// TwinCAT 3 PLC project PLC_2
// ProgramVersion: 3.1.4020.2
// libraries:
//   Tc2_Standard, * (Beckhoff Automation GmbH)
//   Tc2_System, * (Beckhoff Automation GmbH)
//   Tc3_Module, * (Beckhoff Automation GmbH)
// project tree:
//   DUTs/ PALLET.TcDUT
//   / GlobalTextList.TcGTLO, PlcTask.TcTTO, Visualization Manager.TcVMO (not stored)
//   POUs/ MAIN.TcPOU
//   VISUs/ Visualization.TcVIS
// real-time tasks:
//   TASK PlcTask: cycle T#10ms, priority 20, ADS port 350

CONFIGURATION PLC_2
    RESOURCE PLC ON TwinCAT3
        TASK PlcTask(INTERVAL := T#10ms, PRIORITY := 20);
        PROGRAM MAIN WITH PlcTask : MAIN;
    END_RESOURCE
END_CONFIGURATION

// ---- DUTs/PALLET.TcDUT
TYPE PALLET :
STRUCT
	EX : BOOL:=FALSE;
	WS2 : BOOL:=FALSE;
	WS3 : BOOL:=FALSE;
	POSITION : INT:=-1;
	NEXT_PALLET : INT:=0;
	PREVIOUS_PALLET : INT:=0;
	NUMBER : INT;
END_STRUCT
END_TYPE

// ---- POUs/MAIN.TcPOU
PROGRAM MAIN
VAR

PALLETS : ARRAY [1..50] OF PALLET;					// array that will contain the pallet's information. The number of pallets is limitted by 50 but the code work for as many pallets as we want.
INDEX_PALLET : ARRAY [1..50] OF INT := [50(50)];	// array that will contain the index of each pallet in the PALLETS array
NUMBER_PALLETS : ARRAY [1..9] OF INT;				// number of pallets in every possible position of the system

// Inputs
START : BOOL;
P1 : BOOL;
P2 : BOOL;
P3 : BOOL;
L1 : BOOL;
L2 : BOOL;
L3 : BOOL;
PALLET_IN : BOOL;

// Outputs
BA1 : BOOL;
BA2 : BOOL;
BA3 : BOOL;
S1 : BOOL:=TRUE;
S2 : BOOL:=TRUE;
S3 : BOOL:=TRUE;


MOTOR : BOOL;			// Motor signal
COUNTER_IN : INT:=0;	// number of pallets that have been introduced to the system
COUNTER_OUT : INT:=0;	// number of pallets that have been processed by all of th workstation

// Auxiliary variables
STATE_OUT : INT:=0;			
f : INT;
PROCESS_COUNTER_OUT : TON;	// timer 5s
COUNTER_WS2 : TON;			// timer 5s
COUNTER_WS3 : TON;			// timer 5s
COUNTER_PICK2 : TON;		// timer 2s for picking up pallets from conveyor to workstation 2 and timer for letting pallet pass through the stopper 2
COUNTER_PICK3 : TON;		// timer 2s. The same as COUNTER_PICK2 but for workstation 3
COUNTER_PICK1 : TON;		// timer 2s. The same as COUNTER_PICK2 but for workstation 1
POSITION2 : BOOL;			// variable that will indicate that a pallet is in front of workstation 2
POSITION3 : BOOL;			// variable that will indicate that a pallet is in front of workstation 3
POSITION1 : BOOL;			// variable that will indicate that a pallet is in front of workstation 1
INDEX : INT;				// index of the last pallet inside the system

END_VAR


// External states 0, 1, 2 and 3
CASE STATE_OUT OF
	0:
	// state that means that the system is not working
	IF START=TRUE THEN
		STATE_OUT:=1;
		MOTOR:= 1;
	END_IF
	1:
	// system is runing. If we insert a pallet, this state is going to insert the pallet in the system
	IF PALLET_IN=TRUE AND NOT L1 THEN
		STATE_OUT:=2;		
		COUNTER_IN:=COUNTER_IN+1;		
		IF (COUNTER_IN-COUNTER_OUT)>1 THEN
			PALLETS[INDEX].NEXT_PALLET := (COUNTER_IN-COUNTER_OUT);
			PALLETS[(COUNTER_IN-COUNTER_OUT)].NEXT_PALLET :=0;
			PALLETS[(COUNTER_IN-COUNTER_OUT)].PREVIOUS_PALLET :=INDEX;			
		END_IF
		L1:=TRUE;
		PALLET_IN:=FALSE;
		PROCESS_COUNTER_OUT(IN:=FALSE, PT :=T#5S);
	END_IF
	IF PALLET_IN AND L1 THEN
		STATE_OUT:=3;
	END_IF
	
	2:
	// when a pallet is inserted, she is inserted in workstation 1 and this workstation start by processing the pallet. This takes 5 seconds
	PROCESS_COUNTER_OUT(IN:=TRUE, PT :=T#5S);
	IF PROCESS_COUNTER_OUT.Q THEN
		STATE_OUT:=3;
		L1:=FALSE;
		INDEX_PALLET[COUNTER_IN]:=COUNTER_IN-COUNTER_OUT;
		NUMBER_PALLETS[1]:=NUMBER_PALLETS[1]+1;
		PALLETS[(COUNTER_IN-COUNTER_OUT)].POSITION :=0;
		PALLETS[(COUNTER_IN-COUNTER_OUT)].EX :=TRUE;
		PALLETS[(COUNTER_IN-COUNTER_OUT)].NUMBER :=COUNTER_IN;
	END_IF
	
	3:
	// in this state, the system will pass through all of the pallets that are in the system. He will see where are they and, depending on the inputs, he will do something to the pallets.
	IF PALLET_IN THEN
		// if PALLETS_IN is pressed, then we have to jump to external state 1 to insert the pallet.
		STATE_OUT:=1;	
	END_IF	
	
	// these nex lines of code exist to find the pallet that is in the front of all of them
	IF PALLETS[1].PREVIOUS_PALLET>0 THEN
		f:=1;
		WHILE PALLETS[f].PREVIOUS_PALLET>0 DO
			f:=PALLETS[f].PREVIOUS_PALLET;
		END_WHILE
	ELSE
		f:=1;
	END_IF	
	
	// WHILE cycle, where the system will pass through all of the pallets in the system
	WHILE f>0 DO
		INDEX:=f;
		// Internal states
		CASE PALLETS[f].POSITION OF
			0:
			// if the pallets is in state (position) 0, she will have to wait for P2 to be pressed to jump to the next position.
			IF P2 AND NOT POSITION2 THEN
				NUMBER_PALLETS[1]:=NUMBER_PALLETS[1]-1;
				NUMBER_PALLETS[2]:=NUMBER_PALLETS[2]+1;
				PALLETS[f].POSITION:=1;
				POSITION2:=TRUE;
				COUNTER_PICK2(IN:=FALSE, PT :=T#2S);
			END_IF
		
			1:
			// if the pallet is in position 1 (in front of workstation 2) we will have to check if the workstation is free and if the pallet does not have the service from this workstation
			IF NOT L2 AND NOT PALLETS[f].WS2 AND S2 THEN
				// if yes, then the workstation has to pick up the pallet. This takes 2 seconds
				BA2:=TRUE;
				COUNTER_PICK2(IN:=TRUE, PT :=T#2S);
				IF COUNTER_PICK2.Q THEN
					NUMBER_PALLETS[2]:=NUMBER_PALLETS[2]-1;
					NUMBER_PALLETS[8]:=NUMBER_PALLETS[8]+1;
					PALLETS[f].POSITION:=7;
					POSITION2:=FALSE;
					P2:=FALSE;
					BA2:=FALSE;
					L2:=TRUE;
					COUNTER_WS2(IN:=FALSE, PT :=T#5S);
				END_IF				
			ELSE
				// if no, then the stopper 2 should go down, letting the pallet pass. This takes also 2 seconds
				IF L2 OR PALLETS[f].WS2 OR NOT S2 THEN
					S2:=FALSE;
					COUNTER_PICK2(IN:=TRUE, PT :=T#2S);
					IF COUNTER_PICK2.Q THEN
						NUMBER_PALLETS[2]:=NUMBER_PALLETS[2]-1;
						NUMBER_PALLETS[3]:=NUMBER_PALLETS[3]+1;
						PALLETS[f].POSITION:=2;
						S2:=TRUE;
						P2:=FALSE;
						POSITION2:=FALSE;
						// when this happens, this pallet passes in front of the pallet that is being processed by the workstation 2
						// these next lines exist to make that change in the order of the pallets
						IF L2 THEN
							PALLETS[PALLETS[f].PREVIOUS_PALLET].NEXT_PALLET:=PALLETS[f].NEXT_PALLET;
							PALLETS[f].NEXT_PALLET:=PALLETS[f].PREVIOUS_PALLET;
							
							PALLETS[f].PREVIOUS_PALLET:= PALLETS[PALLETS[f].PREVIOUS_PALLET].PREVIOUS_PALLET;
							PALLETS[PALLETS[f].NEXT_PALLET].PREVIOUS_PALLET:=f;
							
							IF PALLETS[f].PREVIOUS_PALLET>0 THEN
								PALLETS[PALLETS[f].PREVIOUS_PALLET].NEXT_PALLET:=f;
							END_IF
							
							IF PALLETS[PALLETS[f].NEXT_PALLET].NEXT_PALLET>0 THEN
								PALLETS[PALLETS[PALLETS[f].NEXT_PALLET].NEXT_PALLET].PREVIOUS_PALLET:=PALLETS[f].NEXT_PALLET;
							END_IF
							
						END_IF
						
					END_IF
				END_IF
			END_IF
			
			2:
			// if the pallet is in position 2, she has to wait for P3 to be pressed to jump to position 3
			IF P3 AND NOT POSITION3 THEN
				NUMBER_PALLETS[3]:=NUMBER_PALLETS[3]-1;
				NUMBER_PALLETS[4]:=NUMBER_PALLETS[4]+1;
				PALLETS[f].POSITION:=3;
				POSITION3:=TRUE;
				COUNTER_PICK3(IN:=FALSE, PT :=T#2S);
			END_IF
			
			3:
			//in this position we have to do the samething that we did in position 1
			IF NOT L3 AND NOT PALLETS[f].WS3 AND S3 THEN
				// if the pallet does not have the service from workstation 3 and this workstation is free, then the pallet goes inside the workstation. This takes 2 seconds
				BA3:=TRUE;
				COUNTER_PICK3(IN:=TRUE, PT :=T#2S);
				IF COUNTER_PICK3.Q THEN
					NUMBER_PALLETS[4]:=NUMBER_PALLETS[4]-1;
					NUMBER_PALLETS[9]:=NUMBER_PALLETS[9]+1;
					PALLETS[f].POSITION:=8;
					BA3:=FALSE;
					P3:=FALSE;
					POSITION3:=FALSE;
					L3:=TRUE;
					COUNTER_WS3(IN:=FALSE, PT :=T#5S);
				END_IF				
			ELSE
				IF L3 OR PALLETS[f].WS3 OR NOT S3 THEN
					// if the workstation is working or the pallet alreafy has this servide, then the stopper 3 goes down and the pallet passes to position 4
					S3:=FALSE;
					COUNTER_PICK3(IN:=TRUE, PT :=T#2S);
					IF COUNTER_PICK3.Q THEN
						NUMBER_PALLETS[4]:=NUMBER_PALLETS[4]-1;
						NUMBER_PALLETS[5]:=NUMBER_PALLETS[5]+1;
						PALLETS[f].POSITION:=4;
						S3:=TRUE;
						P3:=FALSE;
						POSITION3:=FALSE;
						// when this happens, this pallet passes in front of the pallet that is being processed by the workstation 3
						// these next lines exist to make that change in the order of the pallets
						IF L3 THEN
							PALLETS[PALLETS[f].PREVIOUS_PALLET].NEXT_PALLET:=PALLETS[f].NEXT_PALLET;
							PALLETS[f].NEXT_PALLET:=PALLETS[f].PREVIOUS_PALLET;
							
							PALLETS[f].PREVIOUS_PALLET:= PALLETS[PALLETS[f].PREVIOUS_PALLET].PREVIOUS_PALLET;
							PALLETS[PALLETS[f].NEXT_PALLET].PREVIOUS_PALLET:=f;
							
							IF PALLETS[f].PREVIOUS_PALLET>0 THEN
								PALLETS[PALLETS[f].PREVIOUS_PALLET].NEXT_PALLET:=f;
							END_IF
							
							IF PALLETS[PALLETS[f].NEXT_PALLET].NEXT_PALLET>0 THEN
								PALLETS[PALLETS[PALLETS[f].NEXT_PALLET].NEXT_PALLET].PREVIOUS_PALLET:=PALLETS[f].NEXT_PALLET;
							END_IF
							
						END_IF
						
					END_IF
				END_IF
			END_IF
			
			4:
			// in this position, the pallet has to wait for P1 to be pressed to jump to position 5
			IF P1 AND NOT POSITION1 THEN
				NUMBER_PALLETS[5]:=NUMBER_PALLETS[5]-1;
				NUMBER_PALLETS[6]:=NUMBER_PALLETS[6]+1;
				PALLETS[f].POSITION:=5;
				POSITION1:=TRUE;
				COUNTER_PICK1(IN:=FALSE, PT :=T#2S);
			END_IF
			
			5:
			// if the pallet has the service from workstation 2 and 3 and the workstation 1 is free, she is reafy to leave the system. The workstation pickes up the pallet. This takes 2 seconds
			IF NOT L1 AND PALLETS[f].WS3 AND PALLETS[f].WS2 THEN
				BA1:=TRUE;
				COUNTER_PICK1(IN:=TRUE, PT :=T#2S);
				IF COUNTER_PICK1.Q THEN
					NUMBER_PALLETS[6]:=NUMBER_PALLETS[6]-1;
					PALLETS[f].POSITION:=9;
					BA1:=FALSE;
					POSITION1:=FALSE;
					P1:=FALSE;
				END_IF				
			ELSE
				IF L1 OR NOT PALLETS[f].WS3 OR NOT PALLETS[f].WS2 THEN
					// if the pallet does not have the service from workstation 2 or 3 or the workstation is working, then the stopper 1 goes down and the pallet pass to position 0 again.
					S1:=FALSE;
					COUNTER_PICK1(IN:=TRUE, PT :=T#2S);
					IF COUNTER_PICK1.Q THEN
						NUMBER_PALLETS[6]:=NUMBER_PALLETS[6]-1;
						NUMBER_PALLETS[1]:=NUMBER_PALLETS[1]+1;
						PALLETS[f].POSITION:=0;
						S1:=TRUE;
						P1:=FALSE;
						POSITION1:=FALSE;
						// when this happens, this pallet passes in front of the pallet that is being processed by the workstation 1
						// these next lines exist to make that change in the order of the pallets
						IF L1 THEN
							PALLETS[PALLETS[f].PREVIOUS_PALLET].NEXT_PALLET:=PALLETS[f].NEXT_PALLET;
							PALLETS[f].NEXT_PALLET:=PALLETS[f].PREVIOUS_PALLET;
							
							PALLETS[f].PREVIOUS_PALLET:= PALLETS[PALLETS[f].PREVIOUS_PALLET].PREVIOUS_PALLET;
							PALLETS[PALLETS[f].NEXT_PALLET].PREVIOUS_PALLET:=f;
							
							IF PALLETS[f].PREVIOUS_PALLET>0 THEN
								PALLETS[PALLETS[f].PREVIOUS_PALLET].NEXT_PALLET:=f;
							END_IF
							
							IF PALLETS[PALLETS[f].NEXT_PALLET].NEXT_PALLET>0 THEN
								PALLETS[PALLETS[PALLETS[f].NEXT_PALLET].NEXT_PALLET].PREVIOUS_PALLET:=PALLETS[f].NEXT_PALLET;
							END_IF
							
						END_IF
						
					END_IF
				END_IF
			END_IF
			
			7:
			// is the pallet is in position 7, it means that he is being processed by workstation 2. This takes 5 seconds and then the pallet goes to position 2
			COUNTER_WS2(IN:=TRUE, PT :=T#5S);
			IF COUNTER_WS2.Q THEN
				PALLETS[f].WS2:=TRUE;
				L2:=FALSE;
				PALLETS[f].POSITION:=2;
				NUMBER_PALLETS[8]:=NUMBER_PALLETS[8]-1;
				NUMBER_PALLETS[3]:=NUMBER_PALLETS[3]+1;			
				
			END_IF
			
			8:
			// is the pallet is in position 8, it means that he is being processed by workstation 3. This takes 5 seconds and then the pallet goes to position 4
			COUNTER_WS3(IN:=TRUE, PT :=T#5S);
			IF COUNTER_WS3.Q THEN
				NUMBER_PALLETS[9]:=NUMBER_PALLETS[9]-1;
				NUMBER_PALLETS[5]:=NUMBER_PALLETS[5]+1;
				PALLETS[f].POSITION:=4;
				PALLETS[f].WS3:=TRUE;
				L3:=FALSE;
			END_IF
			
			9:
			// if the pallet reach position 9, it means that she has to leave the system. This state has to find where is the pallet in the PALLETS array and then chenge the position of this pallet and the last one. This is going to preserve the free space in the PALLETS array.
			INDEX_PALLET[PALLETS[f].NUMBER]:=50;
			IF f<(COUNTER_IN-COUNTER_OUT) THEN
				INDEX_PALLET[PALLETS[COUNTER_IN-COUNTER_OUT].NUMBER]:=f;
			END_IF
						
			IF (COUNTER_IN-COUNTER_OUT) =1 THEN
				PALLETS[f].PREVIOUS_PALLET:=0;
				PALLETS[f].NEXT_PALLET:=0;
				PALLETS[f].POSITION:=-1;
				PALLETS[f].WS2:=FALSE;
				PALLETS[f].WS3:=FALSE;
				PALLETS[f].EX:=FALSE;
				PALLETS[f].NUMBER:=0;
			ELSE
				IF f=1 THEN
					IF PALLETS[f].NEXT_PALLET>0 THEN
						PALLETS[PALLETS[f].NEXT_PALLET].PREVIOUS_PALLET:=0;
					END_IF										
					IF COUNTER_IN-COUNTER_OUT>2 THEN	
						PALLETS[f].PREVIOUS_PALLET:=COUNTER_IN-COUNTER_OUT-1;					
						PALLETS[COUNTER_IN-COUNTER_OUT-1].NEXT_PALLET:=1;
					ELSE
						PALLETS[f].PREVIOUS_PALLET:=0;
					END_IF
					PALLETS[f].NEXT_PALLET:=0;
					
					PALLETS[f].POSITION:=PALLETS[(COUNTER_IN-COUNTER_OUT)].POSITION;
					PALLETS[f].WS2:=PALLETS[(COUNTER_IN-COUNTER_OUT)].WS2;
					PALLETS[f].WS3:=PALLETS[(COUNTER_IN-COUNTER_OUT)].WS3;
					PALLETS[f].EX:=PALLETS[(COUNTER_IN-COUNTER_OUT)].EX;
					PALLETS[f].NUMBER:=PALLETS[(COUNTER_IN-COUNTER_OUT)].NUMBER;
					
				END_IF
				IF f<(COUNTER_IN-COUNTER_OUT) AND f>1 THEN
					IF PALLETS[f].PREVIOUS_PALLET>0 THEN
						PALLETS[(PALLETS[f].PREVIOUS_PALLET)].NEXT_PALLET:=PALLETS[f].NEXT_PALLET;
					
						IF PALLETS[f].NEXT_PALLET>0 THEN
							PALLETS[(PALLETS[f].NEXT_PALLET)].PREVIOUS_PALLET:=PALLETS[f].PREVIOUS_PALLET;
						END_IF
						PALLETS[PALLETS[COUNTER_IN-COUNTER_OUT].PREVIOUS_PALLET].NEXT_PALLET:=f;
						PALLETS[f].PREVIOUS_PALLET:=PALLETS[COUNTER_IN-COUNTER_OUT].PREVIOUS_PALLET;
						PALLETS[f].NEXT_PALLET:=PALLETS[COUNTER_IN-COUNTER_OUT].NEXT_PALLET;
					ELSE
						PALLETS[(PALLETS[f].NEXT_PALLET)].PREVIOUS_PALLET:=0;
						PALLETS[f].PREVIOUS_PALLET:=PALLETS[COUNTER_IN-COUNTER_OUT].PREVIOUS_PALLET;
						PALLETS[f].NEXT_PALLET:=PALLETS[COUNTER_IN-COUNTER_OUT].NEXT_PALLET;
						PALLETS[PALLETS[COUNTER_IN-COUNTER_OUT].PREVIOUS_PALLET].NEXT_PALLET:=f;
					END_IF					
					
					PALLETS[f].POSITION:=PALLETS[(COUNTER_IN-COUNTER_OUT)].POSITION;
					PALLETS[f].WS2:=PALLETS[(COUNTER_IN-COUNTER_OUT)].WS2;
					PALLETS[f].WS3:=PALLETS[(COUNTER_IN-COUNTER_OUT)].WS3;
					PALLETS[f].EX:=PALLETS[(COUNTER_IN-COUNTER_OUT)].EX;
					PALLETS[f].NUMBER:=PALLETS[(COUNTER_IN-COUNTER_OUT)].NUMBER;							
				END_IF
				IF f=COUNTER_IN-COUNTER_OUT THEN
					PALLETS[COUNTER_IN-COUNTER_OUT-1].NEXT_PALLET:=0;
					IF PALLETS[f].PREVIOUS_PALLET>0 THEN
						PALLETS[PALLETS[f].PREVIOUS_PALLET].NEXT_PALLET:=COUNTER_IN-COUNTER_OUT-1;
					END_IF					
					PALLETS[COUNTER_IN-COUNTER_OUT-1].PREVIOUS_PALLET:= PALLETS[f].PREVIOUS_PALLET;
				END_IF
				PALLETS[(COUNTER_IN-COUNTER_OUT)].POSITION:=-1;
				PALLETS[(COUNTER_IN-COUNTER_OUT)].WS2:=FALSE;
				PALLETS[(COUNTER_IN-COUNTER_OUT)].WS3:=FALSE;
				PALLETS[(COUNTER_IN-COUNTER_OUT)].EX:=FALSE;
				PALLETS[(COUNTER_IN-COUNTER_OUT)].NEXT_PALLET:=0;
				PALLETS[(COUNTER_IN-COUNTER_OUT)].PREVIOUS_PALLET:=0;
				PALLETS[(COUNTER_IN-COUNTER_OUT)].NUMBER:=0;
			END_IF
			COUNTER_OUT:=COUNTER_OUT+1;
			
		END_CASE
		
		f:=PALLETS[f].NEXT_PALLET;
		
	END_WHILE
END_CASE

END_PROGRAM

// ---- GlobalTextList.TcGTLO
TEXTLIST GlobalTextList
  36 = '%s'
  50 = '8'
  51 = '9'
  1 = 'Add pallet'
  20 = 'BA1'
  18 = 'BA2'
  12 = 'BA3'
  32 = 'Behind pallet nº:'
  30 = 'Existence:'
  28 = 'Free'
  33 = 'In front of pallet nº:'
  7 = 'Insert Pallet'
  21 = 'LS1'
  19 = 'LS2'
  13 = 'LS3'
  5 = 'Motor'
  11 = 'Motorstart'
  35 = 'No'
  2 = 'P1'
  3 = 'P2'
  4 = 'P3'
  29 = 'Pallet 1'
  39 = 'Pallet 2'
  42 = 'Pallet 3'
  37 = 'Pallet 4'
  40 = 'Pallet 5'
  43 = 'Pallet 6'
  38 = 'Pallet 7'
  41 = 'Pallet 8'
  44 = 'Pallet 9'
  6 = 'Position 1'
  45 = 'Position 2'
  46 = 'Position 3'
  47 = 'Position 4'
  48 = 'Position 5'
  49 = 'Position 6'
  31 = 'Position:'
  8 = 'Presence 1'
  9 = 'Presence 2'
  10 = 'Presence 3'
  25 = 'PS1'
  14 = 'PS2'
  23 = 'PS3'
  0 = 'Start'
  26 = 'Stopper 1'
  22 = 'Stopper 2'
  24 = 'Stopper 3'
  27 = 'Working'
  17 = 'WS 1'
  16 = 'WS 2'
  15 = 'WS3'
  34 = 'Yes'
END_TEXTLIST

// ---- VISUs/Visualization.TcVIS
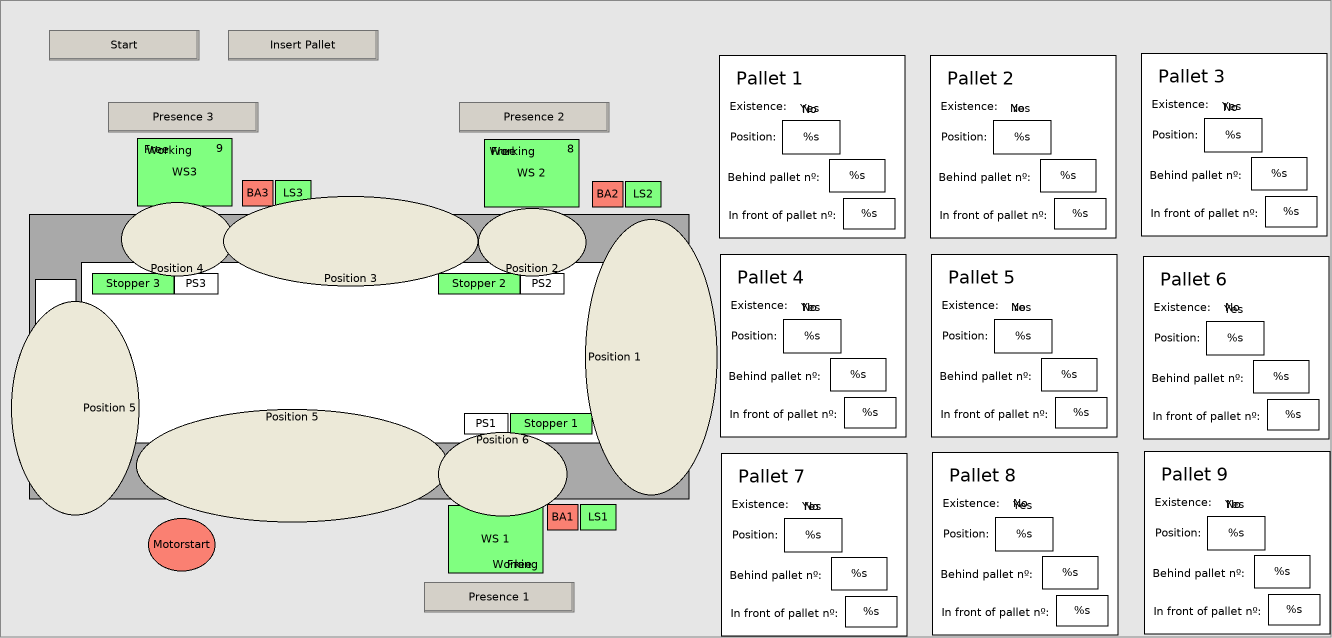
VISUALIZATION Visualization  // 1332x638
    Group (712,55 193x183)
        Rectangle (7,0 186x183)
        Label (14,0 87x47), "Pallet 1"
        Label (0,36 92x31), "Existence:"
        Label (3,65 76x34), "Position:"
        Label (3,111 117x23), "Behind pallet nº:"
        Label (12,147 117x27), "In front of pallet nº:"
        Label (64,34 67x39), "Yes", invisible if: NOT (MAIN.PALLETS[MAIN.INDEX_PALLET[1]].EX)
        Label (64,35 67x39), "No", invisible if: (MAIN.PALLETS[MAIN.INDEX_PALLET[1]].EX)
        Rectangle (70,65 58x34), "%s", text variable: MAIN.PALLETS[MAIN.INDEX_PALLET[1]].POSITION+1
        Rectangle (117,104 56x33), "%s", text variable: MAIN.PALLETS[MAIN.PALLETS[MAIN.INDEX_PALLET[1]].PREVIOUS_PALLET].NUMBER
        Rectangle (131,143 52x31), "%s", text variable: MAIN.PALLETS[MAIN.PALLETS[MAIN.INDEX_PALLET[1]].NEXT_PALLET].NUMBER
    Group (713,254 193x183)
        Rectangle (7,0 186x183)
        Label (14,0 87x47), "Pallet 4"
        Label (0,36 92x31), "Existence:"
        Label (3,65 76x34), "Position:"
        Label (3,111 117x23), "Behind pallet nº:"
        Label (12,147 117x27), "In front of pallet nº:"
        Label (64,34 67x39), "Yes", invisible if: NOT (MAIN.PALLETS[MAIN.INDEX_PALLET[4]].EX)
        Label (63,34 67x39), "No", invisible if: (MAIN.PALLETS[MAIN.INDEX_PALLET[4]].EX)
        Rectangle (70,65 58x34), "%s", text variable: MAIN.PALLETS[MAIN.INDEX_PALLET[4]].POSITION+1
        Rectangle (117,104 56x33), "%s", text variable: MAIN.PALLETS[MAIN.PALLETS[MAIN.INDEX_PALLET[4]].PREVIOUS_PALLET].NUMBER
        Rectangle (131,143 52x31), "%s", text variable: MAIN.PALLETS[MAIN.PALLETS[MAIN.INDEX_PALLET[4]].NEXT_PALLET].NUMBER
    Group (714,453 193x183)
        Rectangle (7,0 186x183)
        Label (14,0 87x47), "Pallet 7"
        Label (0,36 92x31), "Existence:"
        Label (3,65 76x34), "Position:"
        Label (3,111 117x23), "Behind pallet nº:"
        Label (12,147 117x27), "In front of pallet nº:"
        Label (64,34 67x39), "Yes", invisible if: NOT (MAIN.PALLETS[MAIN.INDEX_PALLET[7]].EX)
        Label (64,34 67x39), "No", invisible if: (MAIN.PALLETS[MAIN.INDEX_PALLET[7]].EX)
        Rectangle (70,65 58x34), "%s", text variable: MAIN.PALLETS[MAIN.INDEX_PALLET[7]].POSITION+1
        Rectangle (117,104 56x33), "%s", text variable: MAIN.PALLETS[MAIN.PALLETS[MAIN.INDEX_PALLET[7]].PREVIOUS_PALLET].NUMBER
        Rectangle (131,143 52x31), "%s", text variable: MAIN.PALLETS[MAIN.PALLETS[MAIN.INDEX_PALLET[7]].NEXT_PALLET].NUMBER
    Group (923,55 193x183)
        Rectangle (7,0 186x183)
        Label (14,0 87x47), "Pallet 2"
        Label (0,36 92x31), "Existence:"
        Label (3,65 76x34), "Position:"
        Label (3,111 117x23), "Behind pallet nº:"
        Label (12,147 117x27), "In front of pallet nº:"
        Label (64,34 67x39), "Yes", invisible if: NOT (MAIN.PALLETS[MAIN.INDEX_PALLET[2]].EX)
        Label (61,34 67x39), "No", invisible if: (MAIN.PALLETS[MAIN.INDEX_PALLET[2]].EX)
        Rectangle (70,65 58x34), "%s", text variable: MAIN.PALLETS[MAIN.INDEX_PALLET[2]].POSITION+1
        Rectangle (117,104 56x33), "%s", text variable: MAIN.PALLETS[MAIN.PALLETS[MAIN.INDEX_PALLET[2]].PREVIOUS_PALLET].NUMBER
        Rectangle (131,143 52x31), "%s", text variable: MAIN.PALLETS[MAIN.PALLETS[MAIN.INDEX_PALLET[2]].NEXT_PALLET].NUMBER
    Group (924,254 193x183)
        Rectangle (7,0 186x183)
        Label (14,0 87x47), "Pallet 5"
        Label (0,36 92x31), "Existence:"
        Label (3,65 76x34), "Position:"
        Label (3,111 117x23), "Behind pallet nº:"
        Label (12,147 117x27), "In front of pallet nº:"
        Label (64,34 67x39), "Yes", invisible if: NOT (MAIN.PALLETS[MAIN.INDEX_PALLET[5]].EX)
        Label (61,34 67x39), "No", invisible if: (MAIN.PALLETS[MAIN.INDEX_PALLET[5]].EX)
        Rectangle (70,65 58x34), "%s", text variable: MAIN.PALLETS[MAIN.INDEX_PALLET[5]].POSITION+1
        Rectangle (117,104 56x33), "%s", text variable: MAIN.PALLETS[MAIN.PALLETS[MAIN.INDEX_PALLET[5]].PREVIOUS_PALLET].NUMBER
        Rectangle (131,143 52x31), "%s", text variable: MAIN.PALLETS[MAIN.PALLETS[MAIN.INDEX_PALLET[5]].NEXT_PALLET].NUMBER
    Group (925,452 193x183)
        Rectangle (7,0 186x183)
        Label (14,0 87x47), "Pallet 8"
        Label (0,36 92x31), "Existence:"
        Label (3,65 76x34), "Position:"
        Label (3,111 117x23), "Behind pallet nº:"
        Label (12,147 117x27), "In front of pallet nº:"
        Label (64,34 67x39), "Yes", invisible if: NOT (MAIN.PALLETS[MAIN.INDEX_PALLET[8]].EX)
        Label (62,32 67x39), "No", invisible if: (MAIN.PALLETS[MAIN.INDEX_PALLET[8]].EX)
        Rectangle (70,65 58x34), "%s", text variable: MAIN.PALLETS[MAIN.INDEX_PALLET[8]].POSITION+1
        Rectangle (117,104 56x33), "%s", text variable: MAIN.PALLETS[MAIN.PALLETS[MAIN.INDEX_PALLET[8]].PREVIOUS_PALLET].NUMBER
        Rectangle (131,143 52x31), "%s", text variable: MAIN.PALLETS[MAIN.PALLETS[MAIN.INDEX_PALLET[8]].NEXT_PALLET].NUMBER
    Group (1134,53 193x183)
        Rectangle (7,0 186x183)
        Label (14,0 87x47), "Pallet 3"
        Label (0,36 92x31), "Existence:"
        Label (3,65 76x34), "Position:"
        Label (3,111 117x23), "Behind pallet nº:"
        Label (12,147 117x27), "In front of pallet nº:"
        Label (64,34 67x39), "Yes", invisible if: NOT (MAIN.PALLETS[MAIN.INDEX_PALLET[3]].EX)
        Label (63,35 67x39), "No", invisible if: (MAIN.PALLETS[MAIN.INDEX_PALLET[3]].EX)
        Rectangle (70,65 58x34), "%s", text variable: MAIN.PALLETS[MAIN.INDEX_PALLET[3]].POSITION+1
        Rectangle (117,104 56x33), "%s", text variable: MAIN.PALLETS[MAIN.PALLETS[MAIN.INDEX_PALLET[3]].PREVIOUS_PALLET].NUMBER
        Rectangle (131,143 52x31), "%s", text variable: MAIN.PALLETS[MAIN.PALLETS[MAIN.INDEX_PALLET[3]].NEXT_PALLET].NUMBER
    Group (1136,256 193x183)
        Rectangle (7,0 186x183)
        Label (14,0 87x47), "Pallet 6"
        Label (0,36 92x31), "Existence:"
        Label (3,65 76x34), "Position:"
        Label (3,111 117x23), "Behind pallet nº:"
        Label (12,147 117x27), "In front of pallet nº:"
        Label (64,34 67x39), "Yes", invisible if: NOT (MAIN.PALLETS[MAIN.INDEX_PALLET[6]].EX)
        Label (63,32 67x39), "No", invisible if: (MAIN.PALLETS[MAIN.INDEX_PALLET[6]].EX)
        Rectangle (70,65 58x34), "%s", text variable: MAIN.PALLETS[MAIN.INDEX_PALLET[6]].POSITION+1
        Rectangle (117,104 56x33), "%s", text variable: MAIN.PALLETS[MAIN.PALLETS[MAIN.INDEX_PALLET[6]].PREVIOUS_PALLET].NUMBER
        Rectangle (131,143 52x31), "%s", text variable: MAIN.PALLETS[MAIN.PALLETS[MAIN.INDEX_PALLET[6]].NEXT_PALLET].NUMBER
    Group (1137,451 193x183)
        Rectangle (7,0 186x183)
        Label (14,0 87x47), "Pallet 9"
        Label (0,36 92x31), "Existence:"
        Label (3,65 76x34), "Position:"
        Label (3,111 117x23), "Behind pallet nº:"
        Label (12,147 117x27), "In front of pallet nº:"
        Label (64,34 67x39), "Yes", invisible if: NOT (MAIN.PALLETS[MAIN.INDEX_PALLET[9]].EX)
        Label (63,34 67x39), "No", invisible if: (MAIN.PALLETS[MAIN.INDEX_PALLET[9]].EX)
        Rectangle (70,65 58x34), "%s", text variable: MAIN.PALLETS[MAIN.INDEX_PALLET[9]].POSITION+1
        Rectangle (117,104 56x33), "%s", text variable: MAIN.PALLETS[MAIN.PALLETS[MAIN.INDEX_PALLET[9]].PREVIOUS_PALLET].NUMBER
        Rectangle (131,143 52x31), "%s", text variable: MAIN.PALLETS[MAIN.PALLETS[MAIN.INDEX_PALLET[9]].NEXT_PALLET].NUMBER
    Group (11,30 706x582)
        Group (18,0 660x582)
            Button (20,0 150x30), "Start", colour toggle: MAIN.START
                tap MAIN.START
            Button (199,0 150x30), "Insert Pallet", colour toggle: MAIN.PALLET_IN
                toggle MAIN.PALLET_IN
            Button (395,552 150x30), "Presence 1", colour toggle: MAIN.P1
                toggle MAIN.P1
            Button (430,72 150x30), "Presence 2", colour toggle: MAIN.P2
                toggle MAIN.P2
            Button (79,72 150x30), "Presence 3", colour toggle: MAIN.P3
                toggle MAIN.P3
            RoundedRectangle (0,184 660x285)
            RoundedRectangle (52,232 550x181)
            Ellipse (119,488 67x53), "Motorstart", colour toggle: MAIN.MOTOR
                OnMouseDown: toggle 
            Rectangle (123,189 67x38), invisible if: NOT (MAIN.NUMBER_PALLETS[4]>0)
                OnMouseDown: toggle 
            Rectangle (213,150 31x26), "BA3", colour toggle: MAIN.BA3
                OnMouseDown: toggle 
            Rectangle (246,150 36x26), "LS3", colour toggle: MAIN.L3
                OnMouseDown: toggle 
            Rectangle (491,243 44x21), "PS2", colour toggle: MAIN.P2
                OnMouseDown: toggle 
            Rectangle (108,108 95x68), "WS3", colour toggle: MAIN.L3
                OnMouseDown: toggle 
            Rectangle (455,109 95x68), "WS 2", colour toggle: MAIN.L2
                OnMouseDown: toggle 
            Rectangle (419,475 95x68), "WS 1", colour toggle: MAIN.L1
                OnMouseDown: toggle 
            Rectangle (563,151 31x26), "BA2", colour toggle: MAIN.BA2
                OnMouseDown: toggle 
            Rectangle (596,151 36x26), "LS2", colour toggle: MAIN.L2
                OnMouseDown: toggle 
            Rectangle (518,474 31x26), "BA1", colour toggle: MAIN.BA1
                OnMouseDown: toggle 
            Rectangle (551,474 36x26), "LS1", colour toggle: MAIN.L1
                OnMouseDown: toggle 
            Rectangle (409,243 82x21), "Stopper 2", colour toggle: MAIN.S2
                OnMouseDown: toggle 
            Rectangle (145,243 44x21), "PS3", colour toggle: MAIN.P3
                OnMouseDown: toggle 
            Rectangle (63,243 82x21), "Stopper 3", colour toggle: MAIN.S3
                OnMouseDown: toggle 
            Rectangle (435,383 44x21), "PS1", colour toggle: MAIN.P1
                OnMouseDown: toggle 
            Rectangle (481,383 82x21), "Stopper 1", colour toggle: MAIN.S1
                OnMouseDown: toggle 
            Rectangle (471,189 67x37), invisible if: NOT (MAIN.NUMBER_PALLETS[2]>0)
                OnMouseDown: toggle 
            Rectangle (611,253 41x53), invisible if: NOT (MAIN.NUMBER_PALLETS[1]>=1)
                OnMouseDown: toggle 
            Label (457,524 59x21), "Working", invisible if: NOT MAIN.L1
            Label (454,111 59x21), "Working", invisible if: NOT MAIN.L2
            Label (111,110 59x21), "Working", invisible if: NOT MAIN.L3
            Label (461,524 59x21), "Free", invisible if: MAIN.L1
            Label (445,111 59x21), "Free", invisible if: MAIN.L2
            Label (98,109 59x21), "Free", invisible if: MAIN.L3
            Rectangle (613,315 41x53), invisible if: NOT (MAIN.NUMBER_PALLETS[1]=2)
                OnMouseDown: toggle 
            Rectangle (612,376 41x53), invisible if: NOT (MAIN.NUMBER_PALLETS[1]>2)
                OnMouseDown: toggle 
            Ellipse (630,318 6x4), invisible if: NOT (MAIN.NUMBER_PALLETS[1]>2)
            Ellipse (630,343 6x4), invisible if: NOT (MAIN.NUMBER_PALLETS[1]>2)
            Ellipse (630,357 6x4), invisible if: NOT (MAIN.NUMBER_PALLETS[1]>2)
            Ellipse (630,329 6x4), invisible if: NOT (MAIN.NUMBER_PALLETS[1]>2)
            Rectangle (434,421 67x38), invisible if: NOT (MAIN.NUMBER_PALLETS[6]>0)
                OnMouseDown: toggle 
            Rectangle (230,189 61x37), invisible if: NOT (MAIN.NUMBER_PALLETS[3]>=1)
                OnMouseDown: toggle 
            Rectangle (322,189 60x37), invisible if: NOT (MAIN.NUMBER_PALLETS[3]=2)
                OnMouseDown: toggle 
            Rectangle (370,188 62x38), invisible if: NOT (MAIN.NUMBER_PALLETS[3]>2)
                OnMouseDown: toggle 
            Ellipse (304,207 6x4), invisible if: NOT (MAIN.NUMBER_PALLETS[3]>2)
            Ellipse (325,207 6x4), invisible if: NOT (MAIN.NUMBER_PALLETS[3]>2)
            Ellipse (348,207 6x4), invisible if: NOT (MAIN.NUMBER_PALLETS[3]>2)
            Rectangle (6,249 41x53), invisible if: NOT (MAIN.NUMBER_PALLETS[5]>=1)
                OnMouseDown: toggle 
            Rectangle (6,328 41x53), invisible if: NOT (MAIN.NUMBER_PALLETS[5]=2)
                OnMouseDown: toggle 
            Rectangle (276,418 61x43), invisible if: NOT (MAIN.NUMBER_PALLETS[5]>2)
                OnMouseDown: toggle 
            Ellipse (226,435 6x4), invisible if: NOT (MAIN.NUMBER_PALLETS[5]>2)
            Ellipse (178,435 6x4), invisible if: NOT (MAIN.NUMBER_PALLETS[5]>2)
            Ellipse (127,437 6x4), invisible if: NOT (MAIN.NUMBER_PALLETS[5]>2)
            Ellipse (73,435 6x4), invisible if: NOT (MAIN.NUMBER_PALLETS[5]>2)
            Ellipse (24,393 6x4), invisible if: NOT (MAIN.NUMBER_PALLETS[5]>2)
            Ellipse (23,341 6x4), invisible if: NOT (MAIN.NUMBER_PALLETS[5]>2)
            Ellipse (449,178 108x68), "Position 2"
            Ellipse (92,172 112x74), "Position 4"
            Ellipse (107,379 312x113), "Position 5"
            Ellipse (409,402 129x84), "Position 6"
            Label (527,106 29x26), "8"
            Label (178,108 25x21), "9"
        Ellipse (574,189 132x276), "Position 1"
        Ellipse (212,166 255x90), "Position 3"
        Ellipse (0,271 128x214), "Position 5"
END_VISUALIZATION
